PROGRAM myGun
VAR
	iFiberPres AT %Q* : UINT;
	bFiberOn : BOOL;
	bManualChop : BOOL;
	iFiberScale : UINT;
END_VAR

iFiberScale := PLCSpindleOverride;

IF GVL_IO.bSprayOn = TRUE AND bFiberOn THEN
	iFiberPres :=32000 *iFiberScale/100;
	ELSIF bFiberOn = TRUE AND bManualChop = TRUE THEN
		iFiberPres :=32000*iFiberScale/100;
		ELSE iFiberPres :=0;
END_IF
IF bFiberOn = FALSE THEN
	iFiberPres :=0;
END_IF
IF bManualChop = TRUE AND bFiberOn= TRUE THEN
	iFiberPres :=32000*iFiberScale/100;
END_IF

END_PROGRAM

(* stored: Version 1.1.0.1, ProductVersion 3.1.4024.11
   POU myGun: Id {c52171cb-a448-4d07-a1b3-a884d4516d10}, SpecialFunc None *)
